# EPICS substitutions: exampleTop/DeviceDbApp/UaOpcUaDemoServerDb/UaAnsiCServer.substitutions
file opcuaServerInfo.template {
{ P=$(P=), R=$(R=), SESS=$(SESS) }
}

file opcuaServerStats.template {
{ P=$(P=), R=$(R=), SESS=$(SESS), SUBS=$(SUBS) }
}

file UaOpcUaAnsiCDemoServer.template {
{ P=$(P=), R=$(R=), SESS=$(SESS), SUBS=$(SUBS) }
}
